# EPICS autosave request: motorApp/Db/EnsemblePSOFly_settings.req
$(P)$(Q)startPos
$(P)$(Q)endPos
$(P)$(Q)slewSpeed
$(P)$(Q)scanDelta
$(P)$(Q)detSetupTime
$(P)$(Q)pulseType
$(P)$(Q)scanControl
file calcout_settings.req P=$(P)$(Q)userCalc1
file calcout_settings.req P=$(P)$(Q)userCalc2
file sseq_settings.req P=$(P),S=$(Q)userPreTaxi
file sseq_settings.req P=$(P),S=$(Q)userPreFly
file sseq_settings.req P=$(P),S=$(Q)userPostFly
